Staubli VAL3: onProgEnd.pgx

public program onProgEnd(string& x_sItem[] (dimensions=1))
begin
  //
  // Done, when one program has finished
  //
end
